PROGRAM ControllerMode
VAR_IN_OUT
	fbMover							: MC_PlanarMover;
	fbMover_Axis					: ARRAY [1..6] OF AXIS_REF;
END_VAR
VAR //General
	afbMoverFB						: ARRAY [0..100] OF MC_PlanarFeedback;
	iControlMover					: INT;
	i: INT;
	iCommand: INT;
	
	stActPos						: MoverVector;
	lrStandardPos_x					: LREAL := 120;
	lrStandardPos_y					: LREAL := 120;
	lrStandardPos_c					: LREAL := 0;
END_VAR
VAR //External Set Point
	stExtSetPoi						: ST_ExternalSetpointGenerationOptions;
	stMoverVector_Pos				: MoverVector;
	stMoverVector_Vel				: MoverVector;
	stMoverVector_Acc				: MoverVector;
END_VAR
VAR //Pad
	lrPos_Pad_x						: LREAL;
	lrPos_Pad_y						: LREAL;
	lrPos_Pad_c						: LREAL;
	fbPadPosition					: PositionXYC;
	fbPadCondition					: DynamicConstraint_PathXY;
	bStart_Pad						: BOOL;
	bBusy_Pad						: BOOL;
END_VAR
VAR //Left Stick
	afbMoveAbsolute_LStick_x		: ARRAY [0..1] OF MC_MoveAbsolute;
	afbMoveAbsolute_LStick_y		: ARRAY [0..1] OF MC_MoveAbsolute;
	lrTmpPos_LStick_x				: LREAL;
	lrTmpPos_LStick_y				: LREAL;
	lrPos_LStick_x					: LREAL;
	lrPos_LStick_y					: LREAL;
	lrVel_LStick_x					: LREAL := 500;
	lrVel_LStick_y					: LREAL := 500;
	lrAcc_LStick_x					: LREAL := 1000;
	lrAcc_LStick_y					: LREAL := 1000;
END_VAR
VAR //Right Stick
	lrRange_AB						: LREAL := 1; 
	afbMoveAbsolute_RStick_a		: ARRAY [0..1] OF MC_MoveAbsolute;
	afbMoveAbsolute_RStick_b		: ARRAY [0..1] OF MC_MoveAbsolute;
	lrTmpPos_RStick_a				: LREAL;
	lrTmpPos_RStick_b				: LREAL;
	lrPos_RStick_a					: LREAL;
	lrPos_RStick_b					: LREAL;
	lrVel_RStick_a					: LREAL := 100;
	lrVel_RStick_b					: LREAL := 100;
	lrAcc_RStick_a					: LREAL := 1000;
	lrAcc_RStick_b					: LREAL := 1000;
END_VAR
VAR // A Button
	fbMoveAbsolute_AButton_z		: MC_MoveAbsolute;
	bButton_A						: BOOL;
	bPos_High_z						: BOOL;
	lrPos_AButton_z					: LREAL;
	lrVel_AButton_z					: LREAL := 100;
	lrAcc_AButton_z					: LREAL := 1000;
END_VAR
VAR // B Button
	
END_VAR
VAR // X Button
	
END_VAR
VAR // Y Button
	
END_VAR
VAR //L1 Button
	fbMoveAbsolute_L1Button_c		: MC_MoveAbsolute;
	bButton_L1						: BOOL;
	lrPos_L1Button_c				: LREAL := 200;
	lrVel_L1Button_c				: LREAL := 1000;
	lrAcc_L1Button_c				: LREAL := 10000;
	fbCondition_L1					: DynamicConstraint_Coordinates;
END_VAR
VAR //R1 Button
	fbMoveAbsolute_R1Button_c		: MC_MoveAbsolute;
	bButton_R1						: BOOL;
	lrPos_R1Button_c				: LREAL := 200;
	lrVel_R1Button_c				: LREAL := 1000;
	lrAcc_R1Button_c				: LREAL := 10000;
	fbCondition_R1					: DynamicConstraint_Coordinates;
END_VAR
VAR // L2 Button 
	bReload_L2Button				: BOOL;
	bPosReload_L2Button				: BOOL;
	afbMoveAbsolute_L2Button_c		: ARRAY [0..1] OF MC_MoveAbsolute;
	lrTmpVel_L2Button_c				: LREAL;
	lrPos_L2Button_c				: LREAL;
	lrVel_L2Button_c				: LREAL := 100;
	lrAcc_L2Button_c				: LREAL := 10000;
END_VAR
VAR // R2 Button
	bReload_R2Button				: BOOL;
	bPosReload_R2Button				: BOOL;
	afbMoveAbsolute_R2Button_c		: ARRAY [0..1] OF MC_MoveAbsolute;
	lrTmpVel_R2Button_c				: LREAL;
	lrPos_R2Button_c				: LREAL;
	lrVel_R2Button_c				: LREAL := 100;
	lrAcc_R2Button_c				: LREAL := 10000;
END_VAR
VAR // Start Button
	bPowered						: BOOL;
	bButton_Start					: BOOL;
	afbPower						: ARRAY [1..6] OF MC_Power;
END_VAR
VAR // Back Button
	
END_VAR

stActPos := fbMover.MCTOPLC.ACT.ActPos;

aSystem();
aExternalSetPoint();

FOR i := 0 TO 100 DO
	afbMoverFB[i].Update();
END_FOR

ACTION aCommand:
CASE iCommand OF
	Command.Pad: //十字キー CPosition
	lrPos_Pad_c := stActPos.c;
	fbPadPosition.SetValuesXYC(
		x:= lrPos_Pad_x, y:= lrPos_Pad_y, c:= lrPos_Pad_c);
	fbPadCondition.SetValuesVADJ(
		V:= gc_alrHighCondition_Pos[0], A:= gc_alrHighCondition_Pos[1], 
		D:= gc_alrHighCondition_Pos[2], J:= gc_alrHighCondition_Pos[3]);
	fbMover.MoveToPosition(
		 commandFeedback:= afbMoverFB[2],
		 targetPosition:= fbPadPosition,
		 constraint:= fbPadCondition,
		 options:= 0);
	bBusy_Pad := TRUE;
		
	Command.LeftStick: //XY free move
	IF afbMoveAbsolute_LStick_x[0].Error OR afbMoveAbsolute_LStick_x[1].Error
	OR afbMoveAbsolute_LStick_x[0].Error OR afbMoveAbsolute_LStick_x[1].Error THEN
		afbMoveAbsolute_LStick_x[0].Execute := FALSE;
		afbMoveAbsolute_LStick_x[1].Execute := FALSE;
		afbMoveAbsolute_LStick_y[0].Execute := FALSE;
		afbMoveAbsolute_LStick_y[1].Execute := FALSE;
	END_IF
	//x
	lrTmpPos_LStick_x := lrPos_LStick_x;
	IF g_fbTcJoy.iLeftStick_X_Axis = 0 THEN
		lrPos_LStick_x := 0;
	ELSIF g_fbTcJoy.iLeftStick_X_Axis > 0 THEN 
		lrPos_LStick_x := (g_fbTcJoy.iLeftStick_X_Axis-g_lrDeadZone)/(gc_lrMax_Stick-g_lrDeadZone) * 43;
	ELSE 
		lrPos_LStick_x := (g_fbTcJoy.iLeftStick_X_Axis+g_lrDeadZone)/(gc_lrMax_Stick-g_lrDeadZone) * 43;
	END_IF
	IF lrTmpPos_LStick_x <> lrPos_LStick_x THEN
		IF afbMoveAbsolute_LStick_x[0].Error OR afbMoveAbsolute_LStick_x[1].Error THEN
			afbMoveAbsolute_LStick_x[0].Execute := FALSE;
			afbMoveAbsolute_LStick_x[1].Execute := FALSE;
		ELSIF (NOT afbMoveAbsolute_LStick_x[0].Execute AND NOT afbMoveAbsolute_LStick_x[1].Execute) 
		OR (NOT afbMoveAbsolute_LStick_x[0].Execute AND afbMoveAbsolute_LStick_x[1].Execute) THEN
			afbMoveAbsolute_LStick_x[0].Execute := TRUE;
			afbMoveAbsolute_LStick_x[1].Execute := FALSE;
		ELSE
			afbMoveAbsolute_LStick_x[0].Execute := FALSE;
			afbMoveAbsolute_LStick_x[1].Execute := TRUE;
		END_IF 
	END_IF
	//y
	lrTmpPos_LStick_y := lrPos_LStick_y;
	IF g_fbTcJoy.iLeftStick_Y_Axis = 0 THEN
		lrPos_LStick_y := 0;
	ELSIF g_fbTcJoy.iLeftStick_Y_Axis > 0 THEN
		lrPos_LStick_y := (g_fbTcJoy.iLeftStick_Y_Axis-g_lrDeadZone)/(gc_lrMax_Stick-g_lrDeadZone) * 43;
	ELSE
		lrPos_LStick_y := (g_fbTcJoy.iLeftStick_Y_Axis+g_lrDeadZone)/(gc_lrMax_Stick-g_lrDeadZone) * 43;
	END_IF
	IF lrTmpPos_LStick_y <> lrPos_LStick_y THEN
		IF (NOT afbMoveAbsolute_LStick_y[0].Execute AND NOT afbMoveAbsolute_LStick_y[1].Execute) 
		OR (NOT afbMoveAbsolute_LStick_y[0].Execute AND afbMoveAbsolute_LStick_y[1].Execute) THEN
			afbMoveAbsolute_LStick_y[0].Execute := TRUE;
			afbMoveAbsolute_LStick_y[1].Execute := FALSE;
		ELSE
			afbMoveAbsolute_LStick_y[0].Execute := FALSE;
			afbMoveAbsolute_LStick_y[1].Execute := TRUE;
		END_IF 
	END_IF
	
	FOR i:=0 TO 1 DO
		afbMoveAbsolute_LStick_x[i](
			Axis:= fbMover_Axis[1],
			Position:= lrPos_LStick_x, 
			Velocity:= lrVel_LStick_x, 
			Acceleration:= lrAcc_LStick_x, 
			Deceleration:= lrAcc_LStick_x, 
			Jerk:= lrAcc_LStick_x * 10);
		afbMoveAbsolute_LStick_y[i](
			Axis:= fbMover_Axis[2],
			Position:= lrPos_LStick_y, 
			Velocity:= lrVel_LStick_y, 
			Acceleration:= lrAcc_LStick_y, 
			Deceleration:= lrAcc_LStick_y, 
			Jerk:= lrAcc_LStick_y * 10);
	END_FOR

	Command.RightStick: //AB free move
	IF afbMoveAbsolute_RStick_a[0].Error OR afbMoveAbsolute_RStick_a[1].Error
	OR afbMoveAbsolute_RStick_a[0].Error OR afbMoveAbsolute_RStick_a[1].Error THEN
		afbMoveAbsolute_RStick_a[0].Execute := FALSE;
		afbMoveAbsolute_RStick_a[1].Execute := FALSE;
		afbMoveAbsolute_RStick_b[0].Execute := FALSE;
		afbMoveAbsolute_RStick_b[1].Execute := FALSE;
	END_IF
	IF bPos_High_z THEN
		lrRange_AB := 4;
	ELSE
		lrRange_AB := 1;
	END_IF
	//a
	lrTmpPos_RStick_a := lrPos_RStick_a;
	IF g_fbTcJoy.iRightStick_Y_Axis = 0 THEN
		lrPos_RStick_a := 0;
	ELSIF g_fbTcJoy.iRightStick_Y_Axis > 0 THEN
		lrPos_RStick_a := (g_fbTcJoy.iRightStick_Y_Axis-g_lrDeadZone)/(gc_lrMax_Stick-g_lrDeadZone) * lrRange_AB;
	ELSE
		lrPos_RStick_a := (g_fbTcJoy.iRightStick_Y_Axis+g_lrDeadZone)/(gc_lrMax_Stick-g_lrDeadZone) * lrRange_AB;
	END_IF
	IF lrTmpPos_RStick_a <> lrPos_RStick_a THEN
		IF afbMoveAbsolute_RStick_a[0].Error OR afbMoveAbsolute_RStick_a[1].Error THEN
			afbMoveAbsolute_RStick_a[0].Execute := FALSE;
			afbMoveAbsolute_RStick_a[1].Execute := FALSE;
		ELSIF (NOT afbMoveAbsolute_RStick_a[0].Execute AND NOT afbMoveAbsolute_RStick_a[1].Execute) 
		OR (NOT afbMoveAbsolute_RStick_a[0].Execute AND afbMoveAbsolute_RStick_a[1].Execute) THEN
			afbMoveAbsolute_RStick_a[0].Execute := TRUE;
			afbMoveAbsolute_RStick_a[1].Execute := FALSE;
		ELSE
			afbMoveAbsolute_RStick_a[0].Execute := FALSE;
			afbMoveAbsolute_RStick_a[1].Execute := TRUE;
		END_IF 
	END_IF
	//b
	lrTmpPos_RStick_b := lrPos_RStick_b;
	IF g_fbTcJoy.iRightStick_X_Axis = 0 THEN
		lrPos_RStick_b := 0;
	ELSIF g_fbTcJoy.iRightStick_X_Axis > 0 THEN
		lrPos_RStick_b := (g_fbTcJoy.iRightStick_X_Axis-g_lrDeadZone)/(gc_lrMax_Stick-g_lrDeadZone) * lrRange_AB;
	ELSE
		lrPos_RStick_b := (g_fbTcJoy.iRightStick_X_Axis+g_lrDeadZone)/(gc_lrMax_Stick-g_lrDeadZone) * lrRange_AB;
	END_IF
	IF lrTmpPos_RStick_b <> lrPos_RStick_b THEN
		IF afbMoveAbsolute_RStick_b[0].Error OR afbMoveAbsolute_RStick_b[1].Error THEN
			afbMoveAbsolute_RStick_b[0].Execute := FALSE;
			afbMoveAbsolute_RStick_b[1].Execute := FALSE;
		ELSIF (NOT afbMoveAbsolute_RStick_b[0].Execute AND NOT afbMoveAbsolute_RStick_b[1].Execute) 
		OR (NOT afbMoveAbsolute_RStick_b[0].Execute AND afbMoveAbsolute_RStick_b[1].Execute) THEN
			afbMoveAbsolute_RStick_b[0].Execute := TRUE;
			afbMoveAbsolute_RStick_b[1].Execute := FALSE;
		ELSE
			afbMoveAbsolute_RStick_b[0].Execute := FALSE;
			afbMoveAbsolute_RStick_b[1].Execute := TRUE;
		END_IF 
	END_IF
	
	FOR i:=0 TO 1 DO
		afbMoveAbsolute_RStick_a[i](
			Axis:= fbMover_Axis[4],
			Position:= lrPos_RStick_a, 
			Velocity:= lrVel_RStick_a, 
			Acceleration:= lrAcc_RStick_a, 
			Deceleration:= lrAcc_RStick_a, 
			Jerk:= lrAcc_RStick_a * 10);
		afbMoveAbsolute_RStick_b[i](
			Axis:= fbMover_Axis[5],
			Position:= lrPos_RStick_b, 
			Velocity:= lrVel_RStick_b, 
			Acceleration:= lrAcc_RStick_b, 
			Deceleration:= lrAcc_RStick_b, 
			Jerk:= lrAcc_RStick_b * 10);
	END_FOR
	
	Command.A: // Z Move
	IF bButton_A AND NOT bPos_High_z THEN
		lrPos_AButton_z := 3; //2+3
		fbMoveAbsolute_Abutton_z.Execute := TRUE;
		IF fbMoveAbsolute_Abutton_z.Done OR fbMoveAbsolute_Abutton_z.Error THEN
			fbMoveAbsolute_Abutton_z.Execute := FALSE;
			bButton_A := FALSE;
			bPos_High_z := TRUE;
		END_IF
	ELSIF bButton_A AND bPos_High_z THEN
		lrPos_AButton_z := 0; //2+0
		fbMoveAbsolute_Abutton_z.Execute := TRUE;
		IF fbMoveAbsolute_Abutton_z.Done OR fbMoveAbsolute_Abutton_z.Error THEN
			fbMoveAbsolute_Abutton_z.Execute := FALSE;
			bButton_A := FALSE;
			bPos_High_z := FALSE;
		END_IF
	END_IF
	
	fbMoveAbsolute_Abutton_z(
		Axis:= fbMover_Axis[3],
		Position:= lrPos_AButton_z, 
		Velocity:= lrVel_AButton_z, 
		Acceleration:= lrAcc_AButton_z, 
		Deceleration:= lrAcc_AButton_z, 
		Jerk:= lrAcc_AButton_z * 10);

	Command.B: //Mover Change
	iControlMover := iControlMover +1;

	Command.X: //Mover Change
	iControlMover := iControlMover -1;

	Command.Y: 
		 
	Command.L1: //L1 C CCW 90
	IF bButton_L1 THEN
		lrPos_L1Button_c := lrStandardPos_c + 90;
		fbMoveAbsolute_L1button_c.Execute := TRUE;
		IF fbMoveAbsolute_L1button_c.Done OR fbMoveAbsolute_L1button_c.Error OR fbMoveAbsolute_L1button_c.CommandAborted THEN
			fbMoveAbsolute_L1button_c.Execute := FALSE;
			bButton_L1 := FALSE;
			lrStandardPos_c := lrStandardPos_c + 90;
		END_IF
	END_IF
	fbMoveAbsolute_L1button_c(
		Axis:= fbMover_Axis[6],
		Position:= lrPos_L1Button_c, 
		Velocity:= lrVel_L1Button_c, 
		Acceleration:= lrAcc_L1Button_c, 
		Deceleration:= lrAcc_L1Button_c, 
		Jerk:= lrAcc_L1Button_c * 10);
	
	Command.R1: //R1 C CW 90
	IF bButton_R1 THEN
		lrPos_R1Button_c := lrStandardPos_c - 90;
		fbMoveAbsolute_R1button_c.Execute := TRUE;
		IF fbMoveAbsolute_R1button_c.Done OR fbMoveAbsolute_R1button_c.Error OR fbMoveAbsolute_R1button_c.CommandAborted THEN
			fbMoveAbsolute_R1button_c.Execute := FALSE;
			bButton_R1 := FALSE;
			lrStandardPos_c := lrStandardPos_c - 90;
		END_IF
	END_IF
	fbMoveAbsolute_R1button_c(
		Axis:= fbMover_Axis[6],
		Position:= lrPos_R1Button_c, 
		Velocity:= lrVel_R1Button_c, 
		Acceleration:= lrAcc_R1Button_c, 
		Deceleration:= lrAcc_R1Button_c, 
		Jerk:= lrAcc_R1Button_c * 10);
		
	Command.L2: // Fast C CCW 
	lrTmpVel_L2Button_c := lrVel_L2Button_c;
	IF g_fbTcJoy.iLeftTrigger_Axis = 0 THEN
		afbMoveAbsolute_L2Button_c[0].Execute := FALSE;
		afbMoveAbsolute_L2Button_c[1].Execute := FALSE;
		bPosReload_L2Button := FALSE;
	ELSE
		lrVel_L2Button_c := g_fbTcJoy.iLeftTrigger_Axis/gc_lrMax_L2R2 * 500;
		//更新条件
		IF NOT bPosReload_L2Button AND ABS((lrStandardPos_c-360) - fbMover_Axis[6].NcToPlc.ActPos) < 180 THEN 
			lrStandardPos_c := lrStandardPos_c - 360;
			bPosReload_L2Button := TRUE;
			bReload_L2Button := TRUE;
		ELSIF lrTmpVel_L2Button_c <> lrVel_L2Button_c THEN
			bReload_L2Button := TRUE;
		END_IF
		IF bPosReload_L2Button AND lrStandardPos_c > fbMover_Axis[6].NcToPlc.ActPos THEN
			bPosReload_L2Button := FALSE; 
		END_IF
		
		//更新命令
		IF bReload_L2Button THEN
			bReload_L2Button := FALSE;
			IF (NOT afbMoveAbsolute_L2Button_c[0].Execute AND NOT afbMoveAbsolute_L2Button_c[1].Execute)
			OR (NOT afbMoveAbsolute_L2Button_c[0].Execute AND afbMoveAbsolute_L2Button_c[1].Execute) THEN
				afbMoveAbsolute_L2Button_c[0].Execute := TRUE;
				afbMoveAbsolute_L2Button_c[1].Execute := FALSE;
			ELSE
				afbMoveAbsolute_L2Button_c[0].Execute := FALSE;
				afbMoveAbsolute_L2Button_c[1].Execute := TRUE;
			END_IF
		END_IF
	END_IF
	
	FOR i:=0 TO 1 DO
		lrPos_L2Button_c := lrStandardPos_c - 360;
		afbMoveAbsolute_L2Button_c[i](
			Axis:= fbMover_Axis[6],
			Position:= lrPos_L2Button_c, 
			Velocity:= lrVel_L2Button_c, 
			Acceleration:= lrAcc_L2Button_c, 
			Deceleration:= lrAcc_L2Button_c, 
			Jerk:= lrAcc_L2Button_c * 10);
	END_FOR
	
	Command.R2: // Fast C CW
	lrTmpVel_R2Button_c := lrVel_R2Button_c;
	IF g_fbTcJoy.iRightTrigger_Axis = 0 THEN
		afbMoveAbsolute_R2Button_c[0].Execute := FALSE;
		afbMoveAbsolute_R2Button_c[1].Execute := FALSE;
		bPosReload_R2Button := FALSE;
	ELSE
		lrVel_R2Button_c := g_fbTcJoy.iRightTrigger_Axis/gc_lrMax_L2R2 * 500;
		//更新条件
		IF NOT bPosReload_R2Button AND ABS((lrStandardPos_c+360)  - fbMover_Axis[6].NcToPlc.ActPos) < 180 THEN 
			lrStandardPos_c := lrStandardPos_c + 360;
			bPosReload_R2Button := TRUE;
			bReload_R2Button := TRUE;
		ELSIF lrTmpVel_R2Button_c <> lrVel_R2Button_c THEN
			bReload_R2Button := TRUE;
		END_IF
		IF bPosReload_R2Button AND lrStandardPos_c < fbMover_Axis[6].NcToPlc.ActPos THEN
			bPosReload_R2Button := FALSE; 
		END_IF
		
		//更新命令
		IF bReload_R2Button THEN
			bReload_R2Button := FALSE;
			IF (NOT afbMoveAbsolute_R2Button_c[0].Execute AND NOT afbMoveAbsolute_R2Button_c[1].Execute)
			OR (NOT afbMoveAbsolute_R2Button_c[0].Execute AND afbMoveAbsolute_R2Button_c[1].Execute) THEN
				afbMoveAbsolute_R2Button_c[0].Execute := TRUE;
				afbMoveAbsolute_R2Button_c[1].Execute := FALSE;
			ELSE
				afbMoveAbsolute_R2Button_c[0].Execute := FALSE;
				afbMoveAbsolute_R2Button_c[1].Execute := TRUE;
			END_IF
		END_IF
	END_IF
	
	FOR i:=0 TO 1 DO
		lrPos_R2Button_c := lrStandardPos_c + 360;
		afbMoveAbsolute_R2Button_c[i](
			Axis:= fbMover_Axis[6],
			Position:= lrPos_R2Button_c, 
			Velocity:= lrVel_R2Button_c, 
			Acceleration:= lrAcc_R2Button_c, 
			Deceleration:= lrAcc_R2Button_c, 
			Jerk:= lrAcc_R2Button_c * 10);
	END_FOR
	
	Command.Start: //Servo On Off
	//Power Control
	IF bButton_Start AND bPowered THEN
		fbMover.Disable(commandFeedback:= afbMoverFB[0]);
		IF fbMover.MCTOPLC.STD.State = MC_PLANAR_STATE.Disabled THEN
			bButton_Start := FALSE;
			bPowered := FALSE;
		END_IF
	ELSIF bButton_Start AND NOT bPowered THEN
		fbMover.Enable(commandFeedback:= afbMoverFB[1]);
		IF fbMover.MCTOPLC.STD.State = MC_PLANAR_STATE.Enabled THEN
			bButton_Start := FALSE;
			bPowered := TRUE;
		END_IF
	END_IF

	Command.Back: //Reset
	fbMover.Reset(commandFeedback:= afbMoverFB[5]);
	
END_CASE
END_ACTION

ACTION aExternalSetPoint:
stMoverVector_Pos.x := fbMover_Axis[1].NcToPlc.ActPos;
stMoverVector_Pos.y := fbMover_Axis[2].NcToPlc.ActPos;
stMoverVector_Pos.z := fbMover_Axis[3].NcToPlc.ActPos;
stMoverVector_Pos.a := fbMover_Axis[4].NcToPlc.ActPos;
stMoverVector_Pos.b := fbMover_Axis[5].NcToPlc.ActPos;
stMoverVector_Pos.c := fbMover_Axis[6].NcToPlc.ActPos;

stMoverVector_Vel.x := fbMover_Axis[1].NcToPlc.ActVelo;
stMoverVector_Vel.y := fbMover_Axis[2].NcToPlc.ActVelo;
stMoverVector_Vel.z := fbMover_Axis[3].NcToPlc.ActVelo;
stMoverVector_Vel.a := fbMover_Axis[4].NcToPlc.ActVelo;
stMoverVector_Vel.b := fbMover_Axis[5].NcToPlc.ActVelo;
stMoverVector_Vel.c := fbMover_Axis[6].NcToPlc.ActVelo;

stMoverVector_Acc.x := fbMover_Axis[1].NcToPlc.ActAcc;
stMoverVector_Acc.y := fbMover_Axis[2].NcToPlc.ActAcc;
stMoverVector_Acc.z := fbMover_Axis[3].NcToPlc.ActAcc;
stMoverVector_Acc.a := fbMover_Axis[4].NcToPlc.ActAcc;
stMoverVector_Acc.b := fbMover_Axis[5].NcToPlc.ActAcc;
stMoverVector_Acc.c := fbMover_Axis[6].NcToPlc.ActAcc;
	
IF bPowered AND fbMover.MCTOPLC.STD.State = MC_PLANAR_STATE.Enabled THEN
	fbMover.SetExternalSetpoint(
		setPosition:= stMoverVector_Pos, 
		setVelocity:= stMoverVector_Vel, 
		setAcceleration:= stMoverVector_Acc);
	stExtSetPoi.mode := MC_EXTERNAL_SET_POSITION_MODE.Relative;
	fbMover.StartExternalSetpointGeneration(commandFeedback:= afbMoverFB[5], options:= stExtSetPoi);
ELSE
	fbMover.StopExternalSetpointGeneration(commandFeedback:= afbMoverFB[6]);
END_IF
END_ACTION

ACTION aSystem:
//Error
IF fbMover.MCTOPLC.STD.State = MC_PLANAR_STATE.Error THEN
	iCommand := Command.Back;
	aCommand();
	RETURN;
END_IF

//Power
bButton_Start := g_fbTcJoy.Start_Button OR bButton_Start;
IF bButton_Start THEN
	iCommand := Command.Start;
	aCommand();
	RETURN;
END_IF

IF NOT fbMover.MCTOPLC.STD.State = MC_PLANAR_STATE.Enabled THEN
	RETURN;
END_IF

//Virtual Axis PowerControll
IF bPowered THEN
	FOR i:=1 TO 6 DO
		afbPower[i].Enable := TRUE;
		afbPower[i].Enable_Negative := TRUE;
		afbPower[i].Enable_Positive := TRUE;
		afbPower[i](Axis:=fbMover_Axis[i]);
	END_FOR
ELSE
	FOR i:=1 TO 6 DO
		afbPower[i].Enable := FALSE;
		afbPower[i].Enable_Negative := TRUE;
		afbPower[i].Enable_Positive := TRUE;
		afbPower[i](Axis:=fbMover_Axis[i]);
	END_FOR
END_IF

//Pad
IF NOT bBusy_Pad AND g_fbTcJoy.DPad_Down_Button THEN
	lrPos_Pad_x := lrStandardPos_x;
	lrPos_Pad_y := lrStandardPos_y - 120;
	bStart_Pad := TRUE;
ELSIF NOT bBusy_Pad AND g_fbTcJoy.DPad_Up_Button THEN
	lrPos_Pad_x := lrStandardPos_x;
	lrPos_Pad_y := lrStandardPos_y + 120;
	bStart_Pad := TRUE;
ELSIF NOT bBusy_Pad AND g_fbTcJoy.DPad_Left_Button THEN
	lrPos_Pad_x := lrStandardPos_x - 120;
	lrPos_Pad_y := lrStandardPos_y;
	bStart_Pad := TRUE;
ELSIF NOT bBusy_Pad AND g_fbTcJoy.DPad_Right_Button THEN
	lrPos_Pad_x := lrStandardPos_x + 120;
	lrPos_Pad_y := lrStandardPos_y;
	bStart_Pad := TRUE;
END_IF
IF NOT bBusy_Pad AND bStart_Pad THEN
	iCommand := Command.Pad;
	aCommand();
ELSE
	IF afbMoverFB[2].Done AND bBusy_Pad THEN
		lrStandardPos_x := lrPos_Pad_x;
		lrStandardPos_y := lrPos_Pad_y;
		bBusy_Pad := FALSE;
		bStart_Pad := FALSE;
	ELSIF afbMoverFB[2].Error THEN
		bBusy_Pad := FALSE;
		bStart_Pad := FALSE;
	END_IF
END_IF

//C CCW
bButton_L1 := g_fbTcJoy.LeftShoulder_Button OR bButton_L1;
IF bButton_L1 THEN
	iCommand := Command.L1;
	aCommand();
END_IF


//C CW
bButton_R1 := g_fbTcJoy.RightShoulder_Button OR bButton_R1;
IF bButton_R1 THEN
	iCommand := Command.R1;
	aCommand();
END_IF

//Z
bButton_A := g_fbTcJoy.A_Button OR bButton_A;
IF bButton_A THEN
	iCommand := Command.A;
	aCommand();
END_IF

//L2
iCommand := Command.L2;
aCommand();

//R2
iCommand := Command.R2;
aCommand();

//LStick
iCommand := Command.LeftStick;
aCommand();

//RStick
iCommand := Command.RightStick;
aCommand();
END_ACTION

END_PROGRAM

(* stored: Version 1.1.0.1, ProductVersion 3.1.4024.12
   POU ControllerMode: Id {4c6eba13-5fdf-4d77-bafc-55c67c47bfe1}, SpecialFunc None
   Action aCommand: Id {c01d41ce-d94e-41f6-8bc0-512a9eff8c5d}
   Action aExternalSetPoint: Id {a0bbab1a-2921-467c-b78a-7abc7e4902a1}
   Action aSystem: Id {d64e3794-e70f-4b40-b558-e15566543541} *)
